INTERFACE I_FallibleLREAL EXTENDS I_Fallible

PROPERTY Val : LREAL
GET
END_GET
END_PROPERTY

END_INTERFACE

(* stored: Version 1.1.0.1, ProductVersion 3.1.4022.18
   Itf I_FallibleLREAL: Id {935ca5d4-4e17-467c-a015-f41873a9e1ce}
   Property Val: Id {ba3b5499-970e-4f5a-8ed1-df32fcbe39e1}
   Get Get: Id {0e695ccb-40cb-4691-99c6-84b4bbc769ba} *)
